FUNCTION CopyArray 
VAR_INPUT
	n:INT;	
END_VAR
VAR_IN_OUT
	Source: ARRAY[0..GVL.MaxArraySize]  OF Pancake;
	Target: ARRAY[0..GVL.MaxArraySize]  OF Pancake;
END_VAR
VAR
	i:INT;
END_VAR

FOR i:= 0 TO n DO
	Target[i]:=Source[i];
END_FOR

END_FUNCTION

(* stored: Version 1.1.0.1, ProductVersion 3.1.4022.12
   POU CopyArray: Id {31584b15-9caf-4892-92d4-4fce51d00991}, SpecialFunc None *)
